(* IEC 61131-3 sources: ArfBotOS/Codesys-4/ArfBotOS.fbsdev/Application.iecapp^/FUN/FB_LicenseStatus.fb.st^, 8 files *)

(* ---- FB_LicenseStatus.fb.st ---- *)
FUNCTION_BLOCK FB_LicenseStatus IMPLEMENTS CmpEventMgr.ICmpEventCallback
VAR_OUTPUT
	eState : CmpMgr.RUNTIME_LICENSE_STATE;
	udiSecondsLeft : UDINT;
	udiMinutesLeft : UDINT;
	tRemaining : TIME;
	sState : STRING(32);
	sBanner : STRING(80);
	xDemo : BOOL;
	xLicensed : BOOL;
	xShowBanner : BOOL;
END_VAR
VAR
	_hEvent : SysTypes.RTS_IEC_HANDLE := SysTypes.RTS_INVALID_HANDLE;
	_hCallback : SysTypes.RTS_IEC_HANDLE := SysTypes.RTS_INVALID_HANDLE;
	_result : SysTypes.RTS_IEC_RESULT;
	_xRegistered : BOOL;
	_xTried : BOOL;
	_xGotEvent : BOOL;
	_udiSecondsAtEvent : UDINT;
	_tEvent : TIME;
	_tRetry : TIME;
	_udiElapsed : UDINT;
	_sMin : STRING(11);
	_sSec : STRING(11);
	_udiSec : UDINT;
END_VAR

M_EnsureRegistered();
M_UpdateRemaining();
M_BuildBanner();
END_FUNCTION_BLOCK

(* ---- EventCallback.meth.st ---- *)
METHOD EventCallback : SysTypes.RTS_IEC_RESULT
VAR_INPUT
	pEventParam : POINTER TO CmpEventMgr.EventParam;
END_VAR
VAR
	pLic : POINTER TO CmpMgr.EVTPARAM_CmpMgr_LicenseState;
END_VAR

EventCallback := 0;
IF pEventParam = 0 THEN
	RETURN;
END_IF
IF pEventParam^.EventId <> CmpMgr.EventIDs.EVT_CmpMgr_LicenseState THEN
	RETURN;
END_IF
IF pEventParam^.pParameter = 0 THEN
	RETURN;
END_IF

pLic := pEventParam^.pParameter;
eState := pLic^.state;
_xGotEvent := TRUE;
_tEvent := TIME();
IF pLic^.secondsToExpiration > 0 THEN
	_udiSecondsAtEvent := pLic^.secondsToExpiration;
ELSIF eState = CmpMgr.RUNTIME_LICENSE_STATE.DEMOMODE THEN
	_udiSecondsAtEvent := 7200;
ELSE
	_udiSecondsAtEvent := 0;
END_IF
udiSecondsLeft := _udiSecondsAtEvent;
END_METHOD

(* ---- FB_Exit.meth.st ---- *)
METHOD FB_Exit : BOOL
VAR_INPUT
	bInCopyCode : BOOL;
END_VAR

IF NOT bInCopyCode THEN
	M_Unregister();
END_IF
FB_Exit := TRUE;
END_METHOD

(* ---- FB_Init.meth.st ---- *)
METHOD FB_Init : BOOL
VAR_INPUT
	bInitRetains : BOOL;
	bInCopyCode : BOOL;
END_VAR

IF NOT bInCopyCode THEN
	M_EnsureRegistered();
END_IF
FB_Init := TRUE;
END_METHOD

(* ---- M_BuildBanner.meth.st ---- *)
METHOD PRIVATE M_BuildBanner

CASE eState OF
	CmpMgr.RUNTIME_LICENSE_STATE.DEMOMODE:
		sState := 'DEMO';
	CmpMgr.RUNTIME_LICENSE_STATE.LICENSED:
		sState := 'LICENSED';
	CmpMgr.RUNTIME_LICENSE_STATE.LICENSE_LOST:
		sState := 'LICENSE LOST';
	CmpMgr.RUNTIME_LICENSE_STATE.TRIGGER_SHUTDOWN:
		sState := 'SHUTTING DOWN';
	CmpMgr.RUNTIME_LICENSE_STATE.SAFEMODE:
		sState := 'SAFE MODE';
ELSE
	sState := '';
END_CASE

IF NOT xShowBanner THEN
	sBanner := '';
	RETURN;
END_IF

IF eState = CmpMgr.RUNTIME_LICENSE_STATE.DEMOMODE THEN
	_udiSec := udiSecondsLeft MOD 60;
	_sMin := UDINT_TO_STRING(udiMinutesLeft);
	_sSec := UDINT_TO_STRING(_udiSec);
	sBanner := CONCAT('CODESYS RUNTIME DEMO LICENSE  ', _sMin);
	sBanner := CONCAT(sBanner, 'm ');
	sBanner := CONCAT(sBanner, _sSec);
	sBanner := CONCAT(sBanner, 's remaining');
ELSIF eState = CmpMgr.RUNTIME_LICENSE_STATE.TRIGGER_SHUTDOWN THEN
	sBanner := CONCAT('LICENSE SHUTDOWN  ', UDINT_TO_STRING(udiSecondsLeft));
	sBanner := CONCAT(sBanner, 's');
ELSE
	sBanner := sState;
END_IF
END_METHOD

(* ---- M_EnsureRegistered.meth.st ---- *)
METHOD PRIVATE M_EnsureRegistered
VAR
	tNow : TIME;
END_VAR

IF _xRegistered THEN
	RETURN;
END_IF

tNow := TIME();
IF _xTried AND ((tNow - _tRetry) < T#2S) THEN
	RETURN;
END_IF
_xTried := TRUE;
_tRetry := tNow;

IF _hEvent = SysTypes.RTS_INVALID_HANDLE THEN
	_hEvent := CmpEventMgr.EventOpen(
		EventId := CmpMgr.EventIDs.EVT_CmpMgr_LicenseState,
		CmpIdProvider := CmpMgr.ComponentID.CMPID_CmpMgr,
		Result := _result);
END_IF

IF _hEvent = SysTypes.RTS_INVALID_HANDLE THEN
	RETURN;
END_IF

_hCallback := CmpEventMgr.EventRegisterCallback2(
	hEvent := _hEvent,
	pICallback := THIS^,
	pUserParameter := 0,
	Result := _result);

IF _hCallback <> SysTypes.RTS_INVALID_HANDLE THEN
	_xRegistered := TRUE;
END_IF
END_METHOD

(* ---- M_Unregister.meth.st ---- *)
METHOD PRIVATE M_Unregister

IF _hCallback <> SysTypes.RTS_INVALID_HANDLE THEN
	_result := CmpEventMgr.EventUnregisterCallback(
		hEvent := _hEvent,
		hInterface := _hCallback);
END_IF
IF _hEvent <> SysTypes.RTS_INVALID_HANDLE THEN
	_result := CmpEventMgr.EventClose2(hEvent := _hEvent);
END_IF
_hEvent := SysTypes.RTS_INVALID_HANDLE;
_hCallback := SysTypes.RTS_INVALID_HANDLE;
_xRegistered := FALSE;
END_METHOD

(* ---- M_UpdateRemaining.meth.st ---- *)
METHOD PRIVATE M_UpdateRemaining

xDemo := (eState = CmpMgr.RUNTIME_LICENSE_STATE.DEMOMODE);
xLicensed := (eState = CmpMgr.RUNTIME_LICENSE_STATE.LICENSED);
xShowBanner := xDemo
	OR (eState = CmpMgr.RUNTIME_LICENSE_STATE.LICENSE_LOST)
	OR (eState = CmpMgr.RUNTIME_LICENSE_STATE.TRIGGER_SHUTDOWN)
	OR (eState = CmpMgr.RUNTIME_LICENSE_STATE.SAFEMODE);

IF xLicensed THEN
	udiSecondsLeft := 0;
	udiMinutesLeft := 0;
	tRemaining := T#0S;
	RETURN;
END_IF

IF _xGotEvent AND (xDemo OR (eState = CmpMgr.RUNTIME_LICENSE_STATE.TRIGGER_SHUTDOWN)) THEN
	_udiElapsed := TIME_TO_UDINT(TIME() - _tEvent) / 1000;
	IF _udiElapsed < _udiSecondsAtEvent THEN
		udiSecondsLeft := _udiSecondsAtEvent - _udiElapsed;
	ELSE
		udiSecondsLeft := 0;
	END_IF
END_IF

udiMinutesLeft := udiSecondsLeft / 60;
tRemaining := UDINT_TO_TIME(udiSecondsLeft * 1000);
END_METHOD
